GLOBALCONSTANTS AID_OL (* Output line object attribute ids *)
  (* Standard: 61499-1; Description: Copyright (c) 2023 HR Agrartechnik GmbH This program and the accompanying materials are made available under the terms of the Eclipse Public License 2.0 which is available at https://www.eclipse.org/legal/epl-2.0/ SPDX-License-Identifier: EPL-2.0 *)
  (* Version 1.0, 2026-06-20, Franz Höpfinger, HR Agrartechnik GmbH *)
  PACKAGE isobus::UT::Q::const::AID;
  VAR_GLOBAL CONSTANT
    LINE_ATT : USINT := USINT#1; (* 1: AID_OL_LINE_ATT - Object ID of a Line Attributes object. *)
    WIDTH : USINT := USINT#2; (* 2: AID_OL_WIDTH - Width in pixels. *)
    HEIGHT : USINT := USINT#3; (* 3: AID_OL_HEIGHT - Height in pixels. *)
    LINE_DIR : USINT := USINT#4; (* 4: AID_OL_LINE_DIR - Line direction: 0 = Top-left to bottom-right, 1 = Bottom-left to top-right. *)
  END_VAR
END_GLOBALCONSTANTS
